// TIA Portal V17 export
// export: Created 2024-08-09T12:49:57.2589847Z, ExportSetting WithDefaults, DisplayName Totally Integrated Automation Portal, DisplayVersion V17 Update 7, DisplayName TIA Portal Openness, DisplayVersion V17 Update 7, DisplayName TIA Portal Version Control Interface, DisplayVersion V17, DisplayName STEP 7 Professional, DisplayVersion V17 Update 7, DisplayName STEP 7 Safety, DisplayVersion V17 Update 6, DisplayName WinCC Professional, DisplayVersion V17 Update 7
DATA_BLOCK "CirTrouv"   // DB6
{ S7_Optimized_Access := 'TRUE' }
VERSION : 0.1
// stored: AutoNumber true, DBAccessibleFromOPCUA true, DBAccessibleFromWebserver true, IsOnlyStoredInLoadMemory false, IsRetainMemResEnabled false, IsWriteProtectedInAS false, MemoryReserve 100
   VAR
      Circuits_Trouves { ExternalAccessible := 'False'; ExternalVisible := 'False'; ExternalWritable := 'False'} : Array[0.."Nbr_Circuits", 0.."Nbr_Mob_Circuit"] of Int;
      Cir_Select { ExternalAccessible := 'False'; ExternalVisible := 'False'; ExternalWritable := 'False'} : "S_Circuit";
      Circuit { ExternalAccessible := 'False'; ExternalVisible := 'False'; ExternalWritable := 'False'} : Array[0.."Nbr_Mob_Circuit"] of Int;
   END_VAR
BEGIN
   Circuits_Trouves[0,0..49] := -1;
   Circuits_Trouves[1,0..49] := -1;
   Circuits_Trouves[2,0..49] := -1;
   Circuits_Trouves[3,0..49] := -1;
   Circuits_Trouves[4,0..49] := -1;
   Circuits_Trouves[5,0..49] := -1;
   Circuits_Trouves[6,0..49] := -1;
   Circuits_Trouves[7,0..49] := -1;
   Circuits_Trouves[8,0..49] := -1;
   Circuits_Trouves[9,0..49] := -1;
   Circuits_Trouves[10,0..49] := -1;
   Circuits_Trouves[11,0..49] := -1;
   Circuits_Trouves[12,0..49] := -1;
   Circuits_Trouves[13,0..49] := -1;
   Circuits_Trouves[14,0..49] := -1;
   Circuits_Trouves[15,0..49] := -1;
   Circuits_Trouves[16,0..49] := -1;
   Circuits_Trouves[17,0..49] := -1;
   Circuits_Trouves[18,0..49] := -1;
   Circuits_Trouves[19,0..49] := -1;
   Circuits_Trouves[20,0..49] := -1;
   Circuits_Trouves[21,0..49] := -1;
   Circuits_Trouves[22,0..49] := -1;
   Circuits_Trouves[23,0..49] := -1;
   Circuits_Trouves[24,0..49] := -1;
   Circuits_Trouves[25,0..49] := -1;
   Circuits_Trouves[26,0..49] := -1;
   Circuits_Trouves[27,0..49] := -1;
   Circuits_Trouves[28,0..49] := -1;
   Circuits_Trouves[29,0..49] := -1;
   Cir_Select.Origine := -1;
   Cir_Select.Destination := -1;
END_DATA_BLOCK
